MoveL RelTool (p1,10.000000,14.500000,5.500000,\Rx:=0.000000,\Ry:=0.000000),vel1,zoneval,Extruder\WObj:=Workobject_1;
MoveL RelTool (p1,7.500000,14.500000,5.500000,\Rx:=0.000000,\Ry:=0.000000),vel1,zoneval,Extruder\WObj:=Workobject_1;
MoveL RelTool (p1,5.000000,14.500000,5.500000,\Rx:=0.000000,\Ry:=0.000000),vel1,zoneval,Extruder\WObj:=Workobject_1;
MoveL RelTool (p1,3.000000,15.000000,5.500000,\Rx:=0.000000,\Ry:=-0.000000),vel1,zoneval,Extruder\WObj:=Workobject_1;
MoveL RelTool (p1,5.500000,15.000000,5.500000,\Rx:=0.000000,\Ry:=-0.000000),vel1,zoneval,Extruder\WObj:=Workobject_1;
MoveL RelTool (p1,8.000000,15.000000,5.500000,\Rx:=0.000000,\Ry:=-0.000000),vel1,zoneval,Extruder\WObj:=Workobject_1;
MoveL RelTool (p1,10.500000,15.000000,5.500000,\Rx:=0.000000,\Ry:=-0.000000),vel1,zoneval,Extruder\WObj:=Workobject_1;
MoveL RelTool (p1,13.000000,15.000000,5.500000,\Rx:=0.000000,\Ry:=-0.000000),vel1,zoneval,Extruder\WObj:=Workobject_1;
MoveL RelTool (p1,15.500000,15.000000,5.500000,\Rx:=0.000000,\Ry:=-0.000000),vel1,zoneval,Extruder\WObj:=Workobject_1;
MoveL RelTool (p1,18.000000,15.000000,5.614048,\Rx:=0.000000,\Ry:=-3.081691),vel1,zoneval,Extruder\WObj:=Workobject_1;
MoveL RelTool (p1,20.500000,15.000000,6.707804,\Rx:=0.000000,\Ry:=-9.245066),vel1,zoneval,Extruder\WObj:=Workobject_1;
MoveL RelTool (p1,23.000000,15.000000,9.422764,\Rx:=0.000000,\Ry:=-9.490503),vel1,zoneval,Extruder\WObj:=Workobject_1;
MoveL RelTool (p1,25.500000,15.000000,11.327858,\Rx:=0.000000,\Ry:=-6.584018),vel1,zoneval,Extruder\WObj:=Workobject_1;
MoveL RelTool (p1,28.000000,15.000000,12.618444,\Rx:=0.000000,\Ry:=-5.384296),vel1,zoneval,Extruder\WObj:=Workobject_1;
MoveL RelTool (p1,30.500000,15.000000,13.586392,\Rx:=0.000000,\Ry:=-4.324059),vel1,zoneval,Extruder\WObj:=Workobject_1;
MoveL RelTool (p1,33.000000,15.000000,14.312235,\Rx:=0.000000,\Ry:=-3.332856),vel1,zoneval,Extruder\WObj:=Workobject_1;
MoveL RelTool (p1,35.500000,15.000000,14.840100,\Rx:=0.000000,\Ry:=-2.385490),vel1,zoneval,Extruder\WObj:=Workobject_1;
MoveL RelTool (p1,38.000000,15.000000,15.199032,\Rx:=0.000000,\Ry:=-1.498955),vel1,zoneval,Extruder\WObj:=Workobject_1;
MoveL RelTool (p1,40.500000,15.000000,15.408601,\Rx:=0.000000,\Ry:=-0.638264),vel1,zoneval,Extruder\WObj:=Workobject_1;
MoveL RelTool (p1,43.000000,15.000000,15.481399,\Rx:=0.000000,\Ry:=0.205956),vel1,zoneval,Extruder\WObj:=Workobject_1;
MoveL RelTool (p1,45.500000,15.000000,15.410579,\Rx:=0.000000,\Ry:=1.047110),vel1,zoneval,Extruder\WObj:=Workobject_1;
MoveL RelTool (p1,48.000000,15.000000,15.202916,\Rx:=0.000000,\Ry:=1.929563),vel1,zoneval,Extruder\WObj:=Workobject_1;
MoveL RelTool (p1,50.500000,15.000000,14.821120,\Rx:=0.000000,\Ry:=2.244596),vel1,zoneval,Extruder\WObj:=Workobject_1;
MoveL RelTool (p1,53.000000,15.000000,14.273246,\Rx:=0.000000,\Ry:=2.871157),vel1,zoneval,Extruder\WObj:=Workobject_1;
MoveL RelTool (p1,55.500000,15.000000,13.534442,\Rx:=0.000000,\Ry:=3.972201),vel1,zoneval,Extruder\WObj:=Workobject_1;
MoveL RelTool (p1,58.000000,15.000000,12.561834,\Rx:=0.000000,\Ry:=5.746639),vel1,zoneval,Extruder\WObj:=Workobject_1;
MoveL RelTool (p1,60.500000,15.000000,11.216832,\Rx:=0.000000,\Ry:=7.390876),vel1,zoneval,Extruder\WObj:=Workobject_1;
MoveL RelTool (p1,63.000000,15.000000,9.265661,\Rx:=0.000000,\Ry:=10.572597),vel1,zoneval,Extruder\WObj:=Workobject_1;
MoveL RelTool (p1,65.500000,15.000000,6.601352,\Rx:=0.000000,\Ry:=7.190651),vel1,zoneval,Extruder\WObj:=Workobject_1;
MoveL RelTool (p1,68.000000,15.000000,5.576212,\Rx:=0.000000,\Ry:=1.027235),vel1,zoneval,Extruder\WObj:=Workobject_1;
MoveL RelTool (p1,70.500000,15.000000,5.500000,\Rx:=0.000000,\Ry:=-0.000000),vel1,zoneval,Extruder\WObj:=Workobject_1;
MoveL RelTool (p1,73.000000,15.000000,5.500000,\Rx:=0.000000,\Ry:=-0.000000),vel1,zoneval,Extruder\WObj:=Workobject_1;
MoveL RelTool (p1,75.500000,15.000000,5.500000,\Rx:=0.000000,\Ry:=-0.000000),vel1,zoneval,Extruder\WObj:=Workobject_1;
MoveL RelTool (p1,78.000000,15.000000,5.500000,\Rx:=0.000000,\Ry:=-0.000000),vel1,zoneval,Extruder\WObj:=Workobject_1;
MoveL RelTool (p1,80.500000,15.000000,5.500000,\Rx:=0.000000,\Ry:=-0.000000),vel1,zoneval,Extruder\WObj:=Workobject_1;
MoveL RelTool (p1,82.500000,15.500000,5.500000,\Rx:=0.000000,\Ry:=0.000000),vel1,zoneval,Extruder\WObj:=Workobject_1;
MoveL RelTool (p1,80.000000,15.500000,5.500000,\Rx:=0.000000,\Ry:=0.000000),vel1,zoneval,Extruder\WObj:=Workobject_1;
MoveL RelTool (p1,77.500000,15.500000,5.500000,\Rx:=0.000000,\Ry:=0.000000),vel1,zoneval,Extruder\WObj:=Workobject_1;
MoveL RelTool (p1,75.000000,15.500000,5.500000,\Rx:=0.000000,\Ry:=0.000000),vel1,zoneval,Extruder\WObj:=Workobject_1;
MoveL RelTool (p1,72.500000,15.500000,5.500000,\Rx:=0.000000,\Ry:=0.000000),vel1,zoneval,Extruder\WObj:=Workobject_1;
MoveL RelTool (p1,70.000000,15.500000,5.500000,\Rx:=0.000000,\Ry:=0.000000),vel1,zoneval,Extruder\WObj:=Workobject_1;
MoveL RelTool (p1,67.500000,15.500000,5.696103,\Rx:=0.000000,\Ry:=3.252694),vel1,zoneval,Extruder\WObj:=Workobject_1;
MoveL RelTool (p1,65.000000,15.500000,7.002928,\Rx:=0.000000,\Ry:=9.759467),vel1,zoneval,Extruder\WObj:=Workobject_1;
MoveL RelTool (p1,62.500000,15.500000,9.735076,\Rx:=0.000000,\Ry:=8.879279),vel1,zoneval,Extruder\WObj:=Workobject_1;
MoveL RelTool (p1,60.000000,15.500000,11.544035,\Rx:=0.000000,\Ry:=6.074953),vel1,zoneval,Extruder\WObj:=Workobject_1;
MoveL RelTool (p1,57.500000,15.500000,12.764672,\Rx:=0.000000,\Ry:=4.906952),vel1,zoneval,Extruder\WObj:=Workobject_1;
MoveL RelTool (p1,55.000000,15.500000,13.690789,\Rx:=0.000000,\Ry:=3.858696),vel1,zoneval,Extruder\WObj:=Workobject_1;
MoveL RelTool (p1,52.500000,15.500000,14.387947,\Rx:=0.000000,\Ry:=2.871157),vel1,zoneval,Extruder\WObj:=Workobject_1;
MoveL RelTool (p1,50.000000,15.500000,14.897479,\Rx:=0.000000,\Ry:=1.929563),vel1,zoneval,Extruder\WObj:=Workobject_1;
MoveL RelTool (p1,47.500000,15.500000,15.245728,\Rx:=0.000000,\Ry:=1.047110),vel1,zoneval,Extruder\WObj:=Workobject_1;
MoveL RelTool (p1,45.000000,15.500000,15.449045,\Rx:=0.000000,\Ry:=0.205956),vel1,zoneval,Extruder\WObj:=Workobject_1;
MoveL RelTool (p1,42.500000,15.500000,15.489488,\Rx:=0.000000,\Ry:=-0.143358),vel1,zoneval,Extruder\WObj:=Workobject_1;
MoveL RelTool (p1,40.000000,15.500000,15.383515,\Rx:=0.000000,\Ry:=-0.638264),vel1,zoneval,Extruder\WObj:=Workobject_1;
MoveL RelTool (p1,37.500000,15.500000,15.139895,\Rx:=0.000000,\Ry:=-1.498955),vel1,zoneval,Extruder\WObj:=Workobject_1;
MoveL RelTool (p1,35.000000,15.500000,14.745310,\Rx:=0.000000,\Ry:=-2.385490),vel1,zoneval,Extruder\WObj:=Workobject_1;
MoveL RelTool (p1,32.500000,15.500000,14.178280,\Rx:=0.000000,\Ry:=-3.332856),vel1,zoneval,Extruder\WObj:=Workobject_1;
MoveL RelTool (p1,30.000000,15.500000,13.409743,\Rx:=0.000000,\Ry:=-4.324059),vel1,zoneval,Extruder\WObj:=Workobject_1;
MoveL RelTool (p1,27.500000,15.500000,12.393427,\Rx:=0.000000,\Ry:=-5.384296),vel1,zoneval,Extruder\WObj:=Workobject_1;
MoveL RelTool (p1,25.000000,15.500000,11.016835,\Rx:=0.000000,\Ry:=-7.938887),vel1,zoneval,Extruder\WObj:=Workobject_1;
MoveL RelTool (p1,22.500000,15.500000,8.916676,\Rx:=0.000000,\Ry:=-11.285759),vel1,zoneval,Extruder\WObj:=Workobject_1;
MoveL RelTool (p1,20.000000,15.500000,6.390765,\Rx:=0.000000,\Ry:=-6.482955),vel1,zoneval,Extruder\WObj:=Workobject_1;
MoveL RelTool (p1,17.500000,15.500000,5.549338,\Rx:=0.000000,\Ry:=-1.027233),vel1,zoneval,Extruder\WObj:=Workobject_1;
MoveL RelTool (p1,15.000000,15.500000,5.500000,\Rx:=0.000000,\Ry:=0.000000),vel1,zoneval,Extruder\WObj:=Workobject_1;
MoveL RelTool (p1,12.500000,15.500000,5.500000,\Rx:=0.000000,\Ry:=0.000000),vel1,zoneval,Extruder\WObj:=Workobject_1;
MoveL RelTool (p1,10.000000,15.500000,5.500000,\Rx:=0.000000,\Ry:=0.000000),vel1,zoneval,Extruder\WObj:=Workobject_1;
MoveL RelTool (p1,7.500000,15.500000,5.500000,\Rx:=0.000000,\Ry:=0.000000),vel1,zoneval,Extruder\WObj:=Workobject_1;
MoveL RelTool (p1,5.000000,15.500000,5.500000,\Rx:=0.000000,\Ry:=0.000000),vel1,zoneval,Extruder\WObj:=Workobject_1;
MoveL RelTool (p1,3.000000,16.000000,5.500000,\Rx:=0.000000,\Ry:=0),vel1,zoneval,Extruder\WObj:=Workobject_1;
MoveL RelTool (p1,5.000000,16.000000,5.500000,\Rx:=0.000000,\Ry:=-0.000000),vel1,zoneval,Extruder\WObj:=Workobject_1;
MoveL RelTool (p1,7.500000,16.000000,5.500000,\Rx:=0.000000,\Ry:=-0.000000),vel1,zoneval,Extruder\WObj:=Workobject_1;
MoveL RelTool (p1,10.000000,16.000000,5.500000,\Rx:=0.000000,\Ry:=-0.000000),vel1,zoneval,Extruder\WObj:=Workobject_1;
MoveL RelTool (p1,12.500000,16.000000,5.500000,\Rx:=0.000000,\Ry:=-0.000000),vel1,zoneval,Extruder\WObj:=Workobject_1;
MoveL RelTool (p1,15.000000,16.000000,5.500000,\Rx:=0.000000,\Ry:=-0.000000),vel1,zoneval,Extruder\WObj:=Workobject_1;
MoveL RelTool (p1,17.500000,16.000000,5.549338,\Rx:=0.000000,\Ry:=-1.638714),vel1,zoneval,Extruder\WObj:=Workobject_1;
MoveL RelTool (p1,20.000000,16.000000,6.390765,\Rx:=0.000000,\Ry:=-7.195088),vel1,zoneval,Extruder\WObj:=Workobject_1;
MoveL RelTool (p1,22.500000,16.000000,8.916676,\Rx:=0.000000,\Ry:=-10.077047),vel1,zoneval,Extruder\WObj:=Workobject_1;
MoveL RelTool (p1,25.000000,16.000000,11.016835,\Rx:=0.000000,\Ry:=-7.085230),vel1,zoneval,Extruder\WObj:=Workobject_1;
MoveL RelTool (p1,27.500000,16.000000,12.393427,\Rx:=0.000000,\Ry:=-5.384296),vel1,zoneval,Extruder\WObj:=Workobject_1;
MoveL RelTool (p1,30.000000,16.000000,13.409743,\Rx:=0.000000,\Ry:=-4.324059),vel1,zoneval,Extruder\WObj:=Workobject_1;
MoveL RelTool (p1,32.500000,16.000000,14.178280,\Rx:=0.000000,\Ry:=-3.332856),vel1,zoneval,Extruder\WObj:=Workobject_1;
MoveL RelTool (p1,35.000000,16.000000,14.745310,\Rx:=0.000000,\Ry:=-2.385490),vel1,zoneval,Extruder\WObj:=Workobject_1;
MoveL RelTool (p1,37.500000,16.000000,15.139895,\Rx:=0.000000,\Ry:=-1.498955),vel1,zoneval,Extruder\WObj:=Workobject_1;
MoveL RelTool (p1,40.000000,16.000000,15.383515,\Rx:=0.000000,\Ry:=-0.638264),vel1,zoneval,Extruder\WObj:=Workobject_1;
MoveL RelTool (p1,42.500000,16.000000,15.489488,\Rx:=0.000000,\Ry:=0.205956),vel1,zoneval,Extruder\WObj:=Workobject_1;
MoveL RelTool (p1,45.000000,16.000000,15.449045,\Rx:=0.000000,\Ry:=0.977585),vel1,zoneval,Extruder\WObj:=Workobject_1;
MoveL RelTool (p1,47.500000,16.000000,15.245728,\Rx:=0.000000,\Ry:=1.087548),vel1,zoneval,Extruder\WObj:=Workobject_1;
MoveL RelTool (p1,50.000000,16.000000,14.897479,\Rx:=0.000000,\Ry:=1.929563),vel1,zoneval,Extruder\WObj:=Workobject_1;
MoveL RelTool (p1,52.500000,16.000000,14.387947,\Rx:=0.000000,\Ry:=2.871157),vel1,zoneval,Extruder\WObj:=Workobject_1;
MoveL RelTool (p1,55.000000,16.000000,13.690789,\Rx:=0.000000,\Ry:=3.858696),vel1,zoneval,Extruder\WObj:=Workobject_1;
MoveL RelTool (p1,57.500000,16.000000,12.764672,\Rx:=0.000000,\Ry:=4.906952),vel1,zoneval,Extruder\WObj:=Workobject_1;
MoveL RelTool (p1,60.000000,16.000000,11.544035,\Rx:=0.000000,\Ry:=7.377980),vel1,zoneval,Extruder\WObj:=Workobject_1;
MoveL RelTool (p1,62.500000,16.000000,9.735076,\Rx:=0.000000,\Ry:=9.598425),vel1,zoneval,Extruder\WObj:=Workobject_1;
MoveL RelTool (p1,65.000000,16.000000,7.002928,\Rx:=0.000000,\Ry:=8.615508),vel1,zoneval,Extruder\WObj:=Workobject_1;
MoveL RelTool (p1,67.500000,16.000000,5.696103,\Rx:=0.000000,\Ry:=2.996421),vel1,zoneval,Extruder\WObj:=Workobject_1;
MoveL RelTool (p1,70.000000,16.000000,5.500000,\Rx:=0.000000,\Ry:=-0.000000),vel1,zoneval,Extruder\WObj:=Workobject_1;
MoveL RelTool (p1,72.500000,16.000000,5.500000,\Rx:=0.000000,\Ry:=-0.000000),vel1,zoneval,Extruder\WObj:=Workobject_1;
MoveL RelTool (p1,75.000000,16.000000,5.500000,\Rx:=0.000000,\Ry:=-0.000000),vel1,zoneval,Extruder\WObj:=Workobject_1;
MoveL RelTool (p1,77.500000,16.000000,5.500000,\Rx:=0.000000,\Ry:=-0.000000),vel1,zoneval,Extruder\WObj:=Workobject_1;
MoveL RelTool (p1,80.000000,16.000000,5.500000,\Rx:=0.000000,\Ry:=-0.000000),vel1,zoneval,Extruder\WObj:=Workobject_1;
MoveL RelTool (p1,82.500000,16.000000,5.500000,\Rx:=0.000000,\Ry:=-0.000000),vel1,zoneval,Extruder\WObj:=Workobject_1;






MoveL RelTool (p1,82.500000,16.000000,70.00000,\Rx:=0.000000,\Ry:=0.000000),vel1,z0,Extruder\WObj:=Workobject_1;





ConfL\Off;



    ENDPROC
ENDMODULE
